INTERFACE I_XP_Zone

{attribute 'monitoring':='call'}
PROPERTY AccocietedTrack : I_XP_Track
GET
END_GET
SET
END_SET
END_PROPERTY

{attribute 'monitoring':='call'}
PROPERTY CtsMoversInZone : UINT
GET
END_GET
END_PROPERTY

{attribute 'monitoring':='call'}
PROPERTY EndPositionOnTrack : LREAL
GET
END_GET
SET
END_SET
END_PROPERTY

{attribute 'monitoring':='call'}
PROPERTY HR : HRESULT
GET
END_GET
END_PROPERTY

PROPERTY ListOfMoversToCheck : I_CH_List
SET
END_SET
END_PROPERTY

{attribute 'monitoring':='call'}
PROPERTY MoversInZone : REFERENCE TO ARRAY [0..(CHALET_BaseComponents.BaseParameterlist.MAX_OBJECTS-1)] OF I_XP_Mover_PLC // Return a sorted list of movers in this zone. Index 0 is the mover in Front.
GET
END_GET
END_PROPERTY

{attribute 'monitoring':='call'}
PROPERTY StartPositionOnTrack : LREAL
GET
END_GET
SET
END_SET
END_PROPERTY

END_INTERFACE

(* stored: Version 1.1.0.1, ProductVersion 3.1.4024.12
   Itf I_XP_Zone: Id {f7ed9084-1d91-4a24-afb3-3decf0266b57}
   Property AccocietedTrack: Id {f7873565-85e0-4b90-aee8-bd0f62741bae}
   Get Get: Id {6dc9f28f-67dc-412d-b10c-9bd71499709e}
   Set Set: Id {f3065298-e418-4496-9b24-1547bcc84d48}
   Property CtsMoversInZone: Id {ff8a4ed6-a265-45ae-b945-664463976f7f}
   Get Get: Id {15556529-e025-448d-b13d-c32add93d6c4}
   Property EndPositionOnTrack: Id {b3699955-a9df-4778-ac54-d7089ca9fcb0}
   Get Get: Id {eaf19a27-a36a-44d1-8d17-ab8c8b5b1509}
   Set Set: Id {fe4f214d-9606-4520-a23b-672399df9a11}
   Property HR: Id {089edcd2-a1f6-4d57-98d4-9fb2049afb6f}
   Get Get: Id {baede4dd-5f89-4b1d-a915-cd8f97901eff}
   Property ListOfMoversToCheck: Id {57e9e834-5bb0-4d12-a5bf-dd459a681d0d}
   Set Set: Id {a3eeb9ba-8625-4a4f-a9cd-4778906cfa2c}
   Property MoversInZone: Id {35703c49-aaf7-4aa0-8caf-6cf6ee9e4702}
   Get Get: Id {271dd21b-004a-4367-b9fb-5e73f9ff046f}
   Property StartPositionOnTrack: Id {5db129f3-7ae2-404c-9867-7f10558ddf40}
   Get Get: Id {db7b951c-3c1b-49e8-b029-ce8f57b845ce}
   Set Set: Id {bf9396d4-7ff7-422d-85f2-675d9cfef8ed} *)
